// TIA Portal V18 export
FUNCTION "MainDevTrashBin" : Void   // FC17, LAD
{ S7_Optimized_Access := 'TRUE' }
AUTHOR : HenriP
VERSION : 0.1
// stored: AutoNumber true, IsIECCheckEnabled false, SetENOAutomatically false, UDAEnableTagReadback false
   VAR_TEMP
      AxisFault : Bool;
   END_VAR
BEGIN

REGION Network 2: Initial step
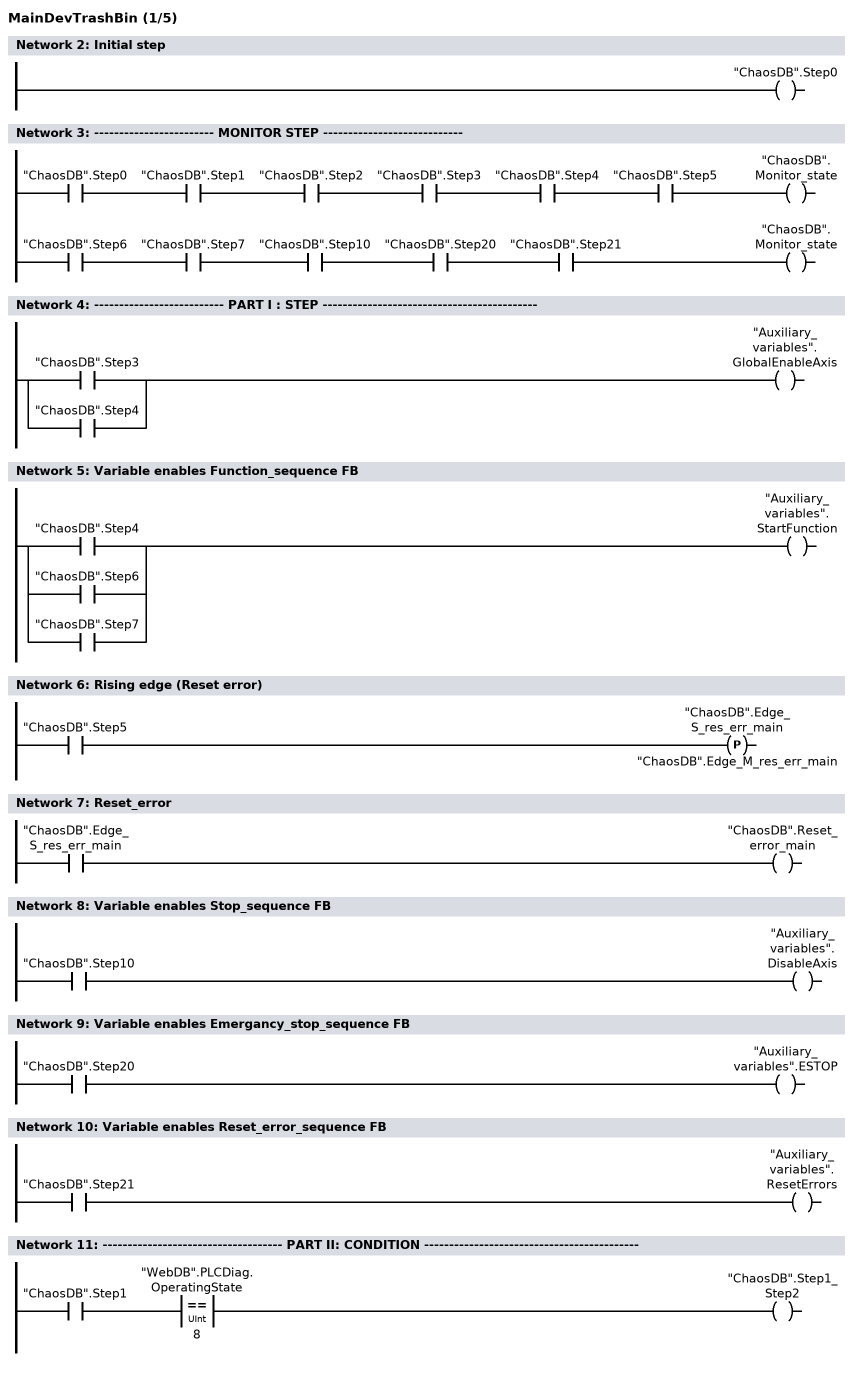
   RUNG wire#powerrail
      Coil( "ChaosDB".Step0 )
   END_RUNG
   // the same network as SCL:
   "ChaosDB".Step0 := TRUE;
END_REGION

REGION Network 3: ------------------------ MONITOR STEP ----------------------------
   RUNG wire#powerrail
      Contact( "ChaosDB".Step0 )
      Contact( "ChaosDB".Step1 )
      Contact( "ChaosDB".Step2 )
      Contact( "ChaosDB".Step3 )
      Contact( "ChaosDB".Step4 )
      Contact( "ChaosDB".Step5 )
      Coil( "ChaosDB".Monitor_state )
   END_RUNG
   RUNG wire#powerrail
      Contact( "ChaosDB".Step6 )
      Contact( "ChaosDB".Step7 )
      Contact( "ChaosDB".Step10 )
      Contact( "ChaosDB".Step20 )
      Contact( "ChaosDB".Step21 )
      Coil( "ChaosDB".Monitor_state )
   END_RUNG
   // the same network as SCL:
   "ChaosDB".Monitor_state := "ChaosDB".Step0 AND "ChaosDB".Step1 AND "ChaosDB".Step2 AND "ChaosDB".Step3 AND "ChaosDB".Step4 AND "ChaosDB".Step5;
   "ChaosDB".Monitor_state := "ChaosDB".Step6 AND "ChaosDB".Step7 AND "ChaosDB".Step10 AND "ChaosDB".Step20 AND "ChaosDB".Step21;
END_REGION

REGION Network 4: -------------------------- PART I : STEP -------------------------------------------
   RUNG wire#powerrail
      Contact( "ChaosDB".Step3 )
      wire#w1
      Coil( "Auxiliary_variables".GlobalEnableAxis )
   END_RUNG
   RUNG wire#powerrail
      Contact( "ChaosDB".Step4 )
   END_RUNG wire#w1
   // the same network as SCL:
   "Auxiliary_variables".GlobalEnableAxis := "ChaosDB".Step3 OR "ChaosDB".Step4;
END_REGION

REGION Network 5: Variable enables Function_sequence FB
   RUNG wire#powerrail
      Contact( "ChaosDB".Step4 )
      wire#w1
      Coil( "Auxiliary_variables".StartFunction )
   END_RUNG
   RUNG wire#powerrail
      Contact( "ChaosDB".Step6 )
   END_RUNG wire#w1
   RUNG wire#powerrail
      Contact( "ChaosDB".Step7 )
   END_RUNG wire#w1
   // the same network as SCL:
   "Auxiliary_variables".StartFunction := "ChaosDB".Step4 OR "ChaosDB".Step6 OR "ChaosDB".Step7;
END_REGION

REGION Network 6: Rising edge (Reset error)
   "ChaosDB".Edge_S_res_err_main := "ChaosDB".Step5 AND NOT "ChaosDB".Edge_M_res_err_main;   // rising edge
   "ChaosDB".Edge_M_res_err_main := "ChaosDB".Step5;
END_REGION

REGION Network 7: Reset_error
   RUNG wire#powerrail
      Contact( "ChaosDB".Edge_S_res_err_main )
      Coil( "ChaosDB".Reset_error_main )
   END_RUNG
   // the same network as SCL:
   "ChaosDB".Reset_error_main := "ChaosDB".Edge_S_res_err_main;
END_REGION

REGION Network 8: Variable enables Stop_sequence FB
   RUNG wire#powerrail
      Contact( "ChaosDB".Step10 )
      Coil( "Auxiliary_variables".DisableAxis )
   END_RUNG
   // the same network as SCL:
   "Auxiliary_variables".DisableAxis := "ChaosDB".Step10;
END_REGION

REGION Network 9: Variable enables Emergancy_stop_sequence FB
   RUNG wire#powerrail
      Contact( "ChaosDB".Step20 )
      Coil( "Auxiliary_variables".ESTOP )
   END_RUNG
   // the same network as SCL:
   "Auxiliary_variables".ESTOP := "ChaosDB".Step20;
END_REGION

REGION Network 10: Variable enables Reset_error_sequence FB
   RUNG wire#powerrail
      Contact( "ChaosDB".Step21 )
      Coil( "Auxiliary_variables".ResetErrors )
   END_RUNG
   // the same network as SCL:
   "Auxiliary_variables".ResetErrors := "ChaosDB".Step21;
END_REGION

REGION Network 11: ------------------------------------ PART II: CONDITION -------------------------------------------
   RUNG wire#powerrail
      Contact( "ChaosDB".Step1 )
      { S7_Templates := "SrcType := UInt" } EQ_Contact(in1 := "WebDB".PLCDiag.OperatingState, in2 := 8)
      Coil( "ChaosDB".Step1_Step2 )
   END_RUNG
   // the same network as SCL:
   "ChaosDB".Step1_Step2 := "ChaosDB".Step1 AND ("WebDB".PLCDiag.OperatingState = 8);
END_REGION

REGION Network 12
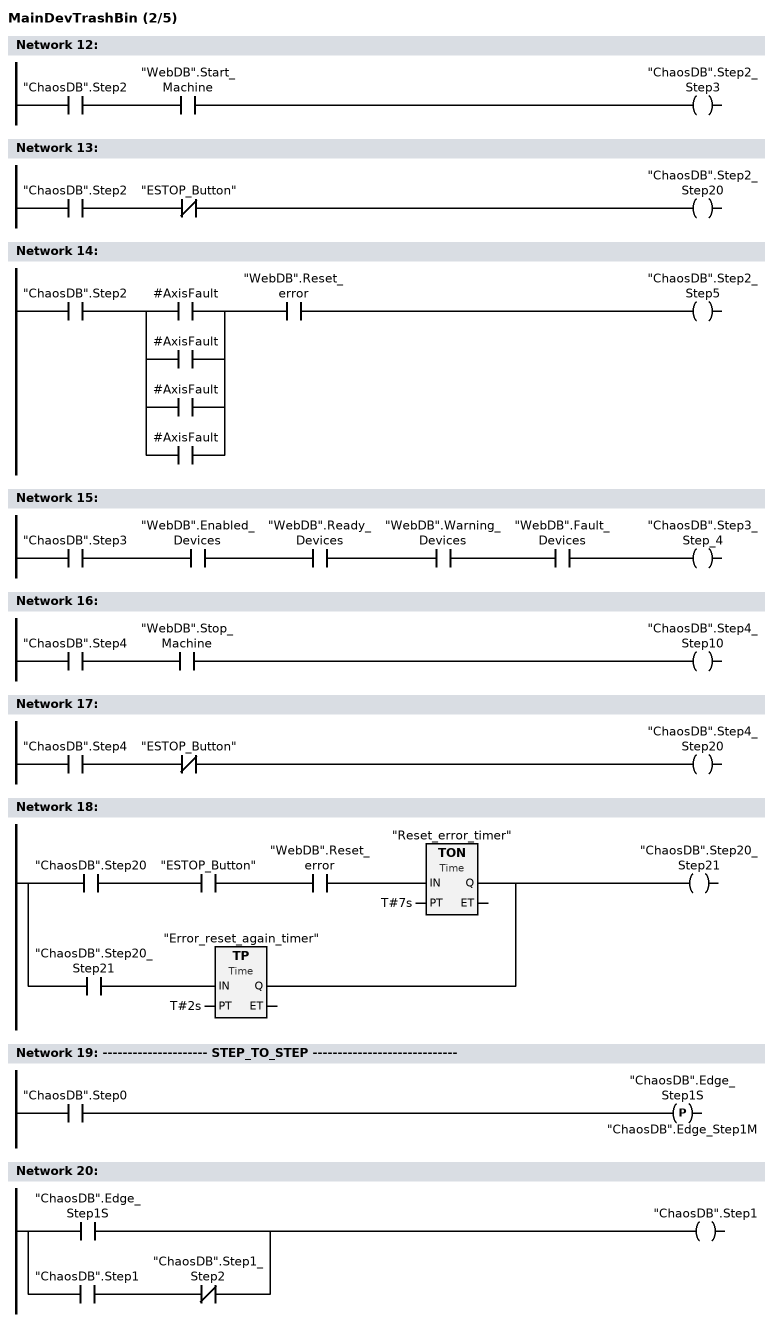
   RUNG wire#powerrail
      Contact( "ChaosDB".Step2 )
      Contact( "WebDB".Start_Machine )
      Coil( "ChaosDB".Step2_Step3 )
   END_RUNG
   // the same network as SCL:
   "ChaosDB".Step2_Step3 := "ChaosDB".Step2 AND "WebDB".Start_Machine;
END_REGION

REGION Network 13
   RUNG wire#powerrail
      Contact( "ChaosDB".Step2 )
      I_Contact( "ESTOP_Button" )
      Coil( "ChaosDB".Step2_Step20 )
   END_RUNG
   // the same network as SCL:
   "ChaosDB".Step2_Step20 := "ChaosDB".Step2 AND NOT "ESTOP_Button";
END_REGION

REGION Network 14
   RUNG wire#powerrail
      Contact( "ChaosDB".Step2 )
      wire#w1
      Contact( #AxisFault )
      wire#w2
      Contact( "WebDB".Reset_error )
      Coil( "ChaosDB".Step2_Step5 )
   END_RUNG
   RUNG wire#w1
      Contact( #AxisFault )
   END_RUNG wire#w2
   RUNG wire#w1
      Contact( #AxisFault )
   END_RUNG wire#w2
   RUNG wire#w1
      Contact( #AxisFault )
   END_RUNG wire#w2
   // the same network as SCL:
   "ChaosDB".Step2_Step5 := "ChaosDB".Step2 AND (#AxisFault OR #AxisFault OR #AxisFault OR #AxisFault) AND "WebDB".Reset_error;
END_REGION

REGION Network 15
   RUNG wire#powerrail
      Contact( "ChaosDB".Step3 )
      Contact( "WebDB".Enabled_Devices )
      Contact( "WebDB".Ready_Devices )
      Contact( "WebDB".Warning_Devices )
      Contact( "WebDB".Fault_Devices )
      Coil( "ChaosDB".Step3_Step_4 )
   END_RUNG
   // the same network as SCL:
   "ChaosDB".Step3_Step_4 := "ChaosDB".Step3 AND "WebDB".Enabled_Devices AND "WebDB".Ready_Devices AND "WebDB".Warning_Devices AND "WebDB".Fault_Devices;
END_REGION

REGION Network 16
   RUNG wire#powerrail
      Contact( "ChaosDB".Step4 )
      Contact( "WebDB".Stop_Machine )
      Coil( "ChaosDB".Step4_Step10 )
   END_RUNG
   // the same network as SCL:
   "ChaosDB".Step4_Step10 := "ChaosDB".Step4 AND "WebDB".Stop_Machine;
END_REGION

REGION Network 17
   RUNG wire#powerrail
      Contact( "ChaosDB".Step4 )
      I_Contact( "ESTOP_Button" )
      Coil( "ChaosDB".Step4_Step20 )
   END_RUNG
   // the same network as SCL:
   "ChaosDB".Step4_Step20 := "ChaosDB".Step4 AND NOT "ESTOP_Button";
END_REGION

REGION Network 18
   RUNG wire#powerrail
      Contact( "ChaosDB".Step20 )
      Contact( "ESTOP_Button" )
      Contact( "WebDB".Reset_error )
      { S7_Templates := "time_type := Time" } "Reset_error_timer".TON(pt := T#7s, et =>)
      wire#w1
      Coil( "ChaosDB".Step20_Step21 )
   END_RUNG
   RUNG wire#powerrail
      Contact( "ChaosDB".Step20_Step21 )
      { S7_Templates := "time_type := Time" } "Error_reset_again_timer".TP(pt := T#2s, et =>)
   END_RUNG wire#w1
   // the same network as SCL:
   "Reset_error_timer".TON(IN := "ChaosDB".Step20 AND "ESTOP_Button" AND "WebDB".Reset_error, PT := T#7s);
   "Error_reset_again_timer".TP(IN := "ChaosDB".Step20_Step21, PT := T#2s);
   "ChaosDB".Step20_Step21 := "Reset_error_timer".Q OR "Error_reset_again_timer".Q;
END_REGION

REGION Network 19: --------------------- STEP_TO_STEP -----------------------------
   "ChaosDB".Edge_Step1S := "ChaosDB".Step0 AND NOT "ChaosDB".Edge_Step1M;   // rising edge
   "ChaosDB".Edge_Step1M := "ChaosDB".Step0;
END_REGION

REGION Network 20
   RUNG wire#powerrail
      Contact( "ChaosDB".Edge_Step1S )
      wire#w1
      Coil( "ChaosDB".Step1 )
   END_RUNG
   RUNG wire#powerrail
      Contact( "ChaosDB".Step1 )
      I_Contact( "ChaosDB".Step1_Step2 )
   END_RUNG wire#w1
   // the same network as SCL:
   "ChaosDB".Step1 := "ChaosDB".Edge_Step1S OR ("ChaosDB".Step1 AND NOT "ChaosDB".Step1_Step2);
END_REGION

REGION Network 21
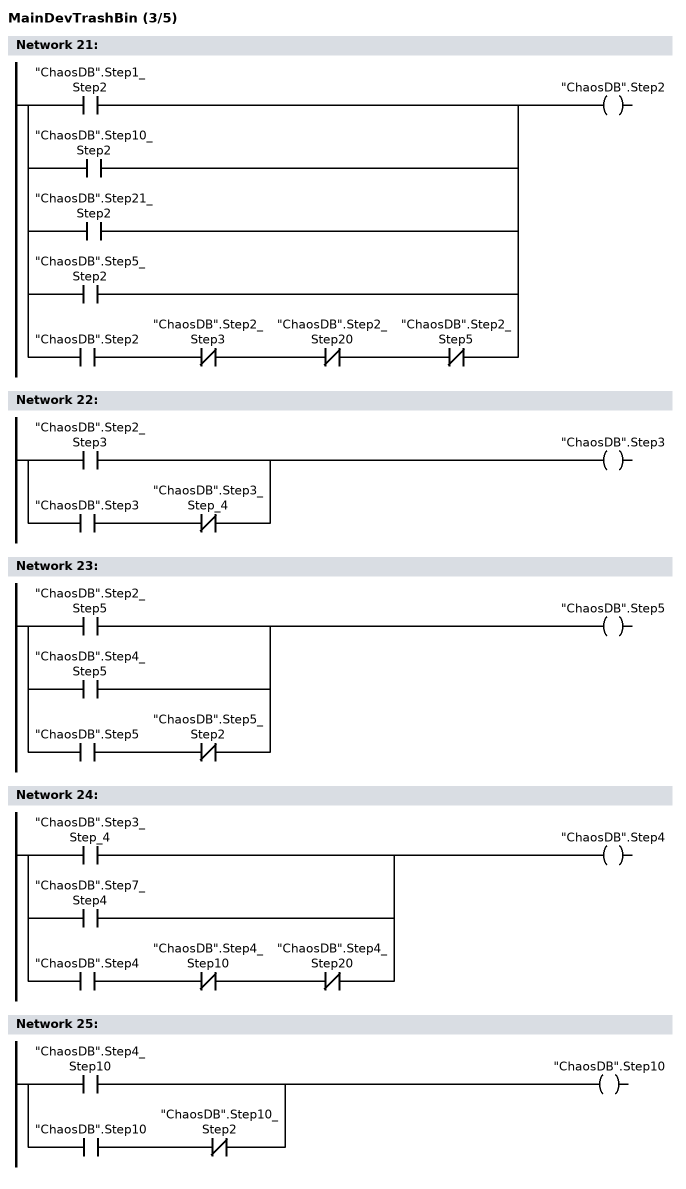
   RUNG wire#powerrail
      Contact( "ChaosDB".Step1_Step2 )
      wire#w1
      Coil( "ChaosDB".Step2 )
   END_RUNG
   RUNG wire#powerrail
      Contact( "ChaosDB".Step10_Step2 )
   END_RUNG wire#w1
   RUNG wire#powerrail
      Contact( "ChaosDB".Step21_Step2 )
   END_RUNG wire#w1
   RUNG wire#powerrail
      Contact( "ChaosDB".Step5_Step2 )
   END_RUNG wire#w1
   RUNG wire#powerrail
      Contact( "ChaosDB".Step2 )
      I_Contact( "ChaosDB".Step2_Step3 )
      I_Contact( "ChaosDB".Step2_Step20 )
      I_Contact( "ChaosDB".Step2_Step5 )
   END_RUNG wire#w1
   // the same network as SCL:
   "ChaosDB".Step2 := "ChaosDB".Step1_Step2 OR "ChaosDB".Step10_Step2 OR "ChaosDB".Step21_Step2 OR "ChaosDB".Step5_Step2 OR ("ChaosDB".Step2 AND NOT "ChaosDB".Step2_Step3 AND NOT "ChaosDB".Step2_Step20 AND NOT "ChaosDB".Step2_Step5);
END_REGION

REGION Network 22
   RUNG wire#powerrail
      Contact( "ChaosDB".Step2_Step3 )
      wire#w1
      Coil( "ChaosDB".Step3 )
   END_RUNG
   RUNG wire#powerrail
      Contact( "ChaosDB".Step3 )
      I_Contact( "ChaosDB".Step3_Step_4 )
   END_RUNG wire#w1
   // the same network as SCL:
   "ChaosDB".Step3 := "ChaosDB".Step2_Step3 OR ("ChaosDB".Step3 AND NOT "ChaosDB".Step3_Step_4);
END_REGION

REGION Network 23
   RUNG wire#powerrail
      Contact( "ChaosDB".Step2_Step5 )
      wire#w1
      Coil( "ChaosDB".Step5 )
   END_RUNG
   RUNG wire#powerrail
      Contact( "ChaosDB".Step4_Step5 )
   END_RUNG wire#w1
   RUNG wire#powerrail
      Contact( "ChaosDB".Step5 )
      I_Contact( "ChaosDB".Step5_Step2 )
   END_RUNG wire#w1
   // the same network as SCL:
   "ChaosDB".Step5 := "ChaosDB".Step2_Step5 OR "ChaosDB".Step4_Step5 OR ("ChaosDB".Step5 AND NOT "ChaosDB".Step5_Step2);
END_REGION

REGION Network 24
   RUNG wire#powerrail
      Contact( "ChaosDB".Step3_Step_4 )
      wire#w1
      Coil( "ChaosDB".Step4 )
   END_RUNG
   RUNG wire#powerrail
      Contact( "ChaosDB".Step7_Step4 )
   END_RUNG wire#w1
   RUNG wire#powerrail
      Contact( "ChaosDB".Step4 )
      I_Contact( "ChaosDB".Step4_Step10 )
      I_Contact( "ChaosDB".Step4_Step20 )
   END_RUNG wire#w1
   // the same network as SCL:
   "ChaosDB".Step4 := "ChaosDB".Step3_Step_4 OR "ChaosDB".Step7_Step4 OR ("ChaosDB".Step4 AND NOT "ChaosDB".Step4_Step10 AND NOT "ChaosDB".Step4_Step20);
END_REGION

REGION Network 25
   RUNG wire#powerrail
      Contact( "ChaosDB".Step4_Step10 )
      wire#w1
      Coil( "ChaosDB".Step10 )
   END_RUNG
   RUNG wire#powerrail
      Contact( "ChaosDB".Step10 )
      I_Contact( "ChaosDB".Step10_Step2 )
   END_RUNG wire#w1
   // the same network as SCL:
   "ChaosDB".Step10 := "ChaosDB".Step4_Step10 OR ("ChaosDB".Step10 AND NOT "ChaosDB".Step10_Step2);
END_REGION

REGION Network 26
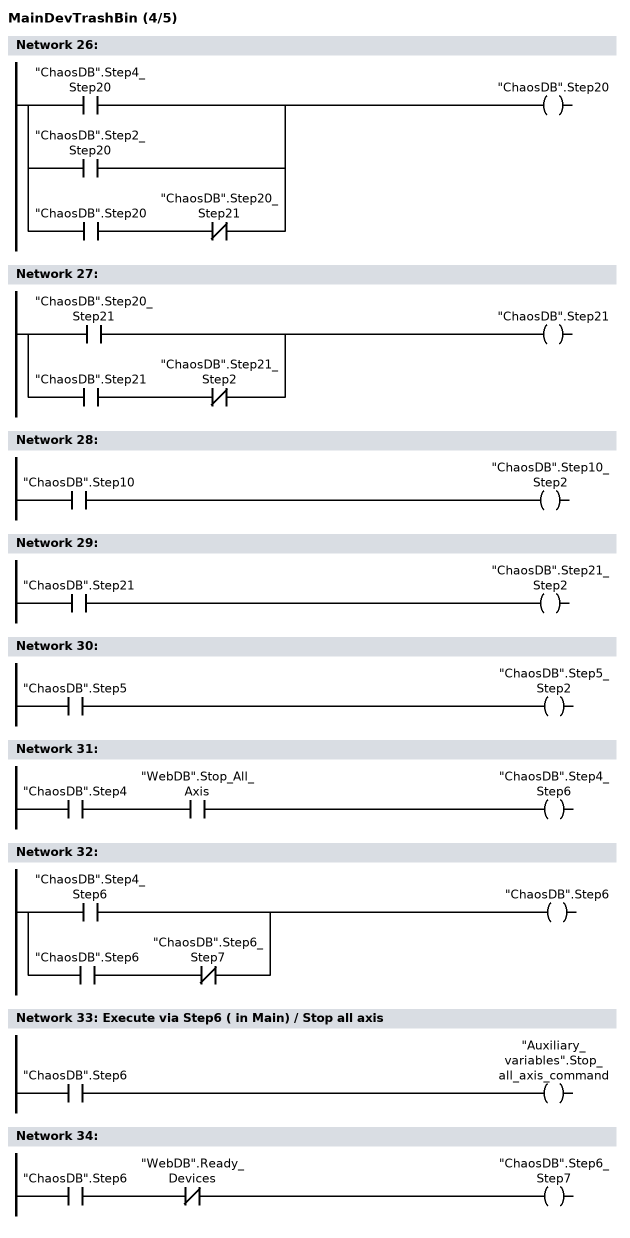
   RUNG wire#powerrail
      Contact( "ChaosDB".Step4_Step20 )
      wire#w1
      Coil( "ChaosDB".Step20 )
   END_RUNG
   RUNG wire#powerrail
      Contact( "ChaosDB".Step2_Step20 )
   END_RUNG wire#w1
   RUNG wire#powerrail
      Contact( "ChaosDB".Step20 )
      I_Contact( "ChaosDB".Step20_Step21 )
   END_RUNG wire#w1
   // the same network as SCL:
   "ChaosDB".Step20 := "ChaosDB".Step4_Step20 OR "ChaosDB".Step2_Step20 OR ("ChaosDB".Step20 AND NOT "ChaosDB".Step20_Step21);
END_REGION

REGION Network 27
   RUNG wire#powerrail
      Contact( "ChaosDB".Step20_Step21 )
      wire#w1
      Coil( "ChaosDB".Step21 )
   END_RUNG
   RUNG wire#powerrail
      Contact( "ChaosDB".Step21 )
      I_Contact( "ChaosDB".Step21_Step2 )
   END_RUNG wire#w1
   // the same network as SCL:
   "ChaosDB".Step21 := "ChaosDB".Step20_Step21 OR ("ChaosDB".Step21 AND NOT "ChaosDB".Step21_Step2);
END_REGION

REGION Network 28
   RUNG wire#powerrail
      Contact( "ChaosDB".Step10 )
      Coil( "ChaosDB".Step10_Step2 )
   END_RUNG
   // the same network as SCL:
   "ChaosDB".Step10_Step2 := "ChaosDB".Step10;
END_REGION

REGION Network 29
   RUNG wire#powerrail
      Contact( "ChaosDB".Step21 )
      Coil( "ChaosDB".Step21_Step2 )
   END_RUNG
   // the same network as SCL:
   "ChaosDB".Step21_Step2 := "ChaosDB".Step21;
END_REGION

REGION Network 30
   RUNG wire#powerrail
      Contact( "ChaosDB".Step5 )
      Coil( "ChaosDB".Step5_Step2 )
   END_RUNG
   // the same network as SCL:
   "ChaosDB".Step5_Step2 := "ChaosDB".Step5;
END_REGION

REGION Network 31
   RUNG wire#powerrail
      Contact( "ChaosDB".Step4 )
      Contact( "WebDB".Stop_All_Axis )
      Coil( "ChaosDB".Step4_Step6 )
   END_RUNG
   // the same network as SCL:
   "ChaosDB".Step4_Step6 := "ChaosDB".Step4 AND "WebDB".Stop_All_Axis;
END_REGION

REGION Network 32
   RUNG wire#powerrail
      Contact( "ChaosDB".Step4_Step6 )
      wire#w1
      Coil( "ChaosDB".Step6 )
   END_RUNG
   RUNG wire#powerrail
      Contact( "ChaosDB".Step6 )
      I_Contact( "ChaosDB".Step6_Step7 )
   END_RUNG wire#w1
   // the same network as SCL:
   "ChaosDB".Step6 := "ChaosDB".Step4_Step6 OR ("ChaosDB".Step6 AND NOT "ChaosDB".Step6_Step7);
END_REGION

REGION Network 33: Execute via Step6 ( in Main) / Stop all axis
   RUNG wire#powerrail
      Contact( "ChaosDB".Step6 )
      Coil( "Auxiliary_variables".Stop_all_axis_command )
   END_RUNG
   // the same network as SCL:
   "Auxiliary_variables".Stop_all_axis_command := "ChaosDB".Step6;
END_REGION

REGION Network 34
   RUNG wire#powerrail
      Contact( "ChaosDB".Step6 )
      I_Contact( "WebDB".Ready_Devices )
      Coil( "ChaosDB".Step6_Step7 )
   END_RUNG
   // the same network as SCL:
   "ChaosDB".Step6_Step7 := "ChaosDB".Step6 AND NOT "WebDB".Ready_Devices;
END_REGION

REGION Network 35
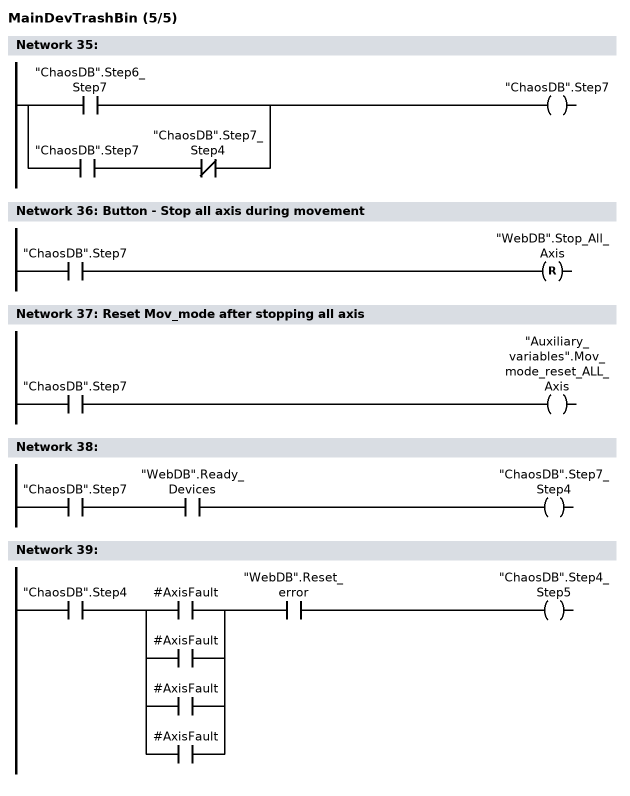
   RUNG wire#powerrail
      Contact( "ChaosDB".Step6_Step7 )
      wire#w1
      Coil( "ChaosDB".Step7 )
   END_RUNG
   RUNG wire#powerrail
      Contact( "ChaosDB".Step7 )
      I_Contact( "ChaosDB".Step7_Step4 )
   END_RUNG wire#w1
   // the same network as SCL:
   "ChaosDB".Step7 := "ChaosDB".Step6_Step7 OR ("ChaosDB".Step7 AND NOT "ChaosDB".Step7_Step4);
END_REGION

REGION Network 36: Button - Stop all axis during movement
   RUNG wire#powerrail
      Contact( "ChaosDB".Step7 )
      R_Coil( "WebDB".Stop_All_Axis )
   END_RUNG
   // the same network as SCL:
   IF "ChaosDB".Step7 THEN "WebDB".Stop_All_Axis := FALSE; END_IF;
END_REGION

REGION Network 37: Reset Mov_mode after stopping all axis
   RUNG wire#powerrail
      Contact( "ChaosDB".Step7 )
      Coil( "Auxiliary_variables".Mov_mode_reset_ALL_Axis )
   END_RUNG
   // the same network as SCL:
   "Auxiliary_variables".Mov_mode_reset_ALL_Axis := "ChaosDB".Step7;
END_REGION

REGION Network 38
   RUNG wire#powerrail
      Contact( "ChaosDB".Step7 )
      Contact( "WebDB".Ready_Devices )
      Coil( "ChaosDB".Step7_Step4 )
   END_RUNG
   // the same network as SCL:
   "ChaosDB".Step7_Step4 := "ChaosDB".Step7 AND "WebDB".Ready_Devices;
END_REGION

REGION Network 39
   RUNG wire#powerrail
      Contact( "ChaosDB".Step4 )
      wire#w1
      Contact( #AxisFault )
      wire#w2
      Contact( "WebDB".Reset_error )
      Coil( "ChaosDB".Step4_Step5 )
   END_RUNG
   RUNG wire#w1
      Contact( #AxisFault )
   END_RUNG wire#w2
   RUNG wire#w1
      Contact( #AxisFault )
   END_RUNG wire#w2
   RUNG wire#w1
      Contact( #AxisFault )
   END_RUNG wire#w2
   // the same network as SCL:
   "ChaosDB".Step4_Step5 := "ChaosDB".Step4 AND (#AxisFault OR #AxisFault OR #AxisFault OR #AxisFault) AND "WebDB".Reset_error;
END_REGION
END_FUNCTION
